Staubli VAL3: Day4.dtx

string sInput
lists lResult
  [0]
    string sString
num nResult
table tTable
  [0]
    num nMatrix[1 1]
lists lLine
  [0]
    string sString
num nBingoNumbers1
num nBingoNumbers2
num nBingoNumbers
table tTable_remove
  [0]
    num nMatrix[1 1]
table tTable_empty
  [0]
    num nMatrix[1 1]
num nResultRow
num nResultCol
bool bWinner
num nIndexX
num nIndexY
bool bFound
bool bHasWon
